Staubli VAL3: refreshProg.pgx

program refreshProg(progItem& x_pProg[])
  local num i
  local num l_nSize
  local string l_sEvent
  local string l_sTitle
  local progItem l_pProg
  local string l_sData
begin
  // set the size of the windows
  if !(cycleStatus:bTraj)
    call use:setView(bLarge)
  endIf
  // Create the list
  if bLarge
    call use:type(2,0,sProgName)
  else
    call use:type(21,0,sProgName)
  endIf
  // fill IT
  call use:listempty()
  if sProgName!=""
    l_nSize=size(x_pProg.iEvent)
    for i=0 to l_nSize-1
      l_nSize=size(x_pProg.iEvent)
      // insert all
      if i<=size(x_pProg.iEvent)-1
        l_sData=x_pProg.iEvent[min(i,size(x_pProg.iEvent)-1)].sData
        l_sEvent=x_pProg.iEvent[min(i,size(x_pProg.iEvent)-1)].sType
        call saveInputOutput:replaceIO(l_sData,l_sEvent,l_sData)
        l_sEvent=l_sEvent+" "+l_sData
        l_sEvent=toString("2",i+1)+" "+l_sEvent
        call use:listadd(l_sEvent)
      else
        return
      endIf
    endFor
  endIf
end
